          TagStructureMember "nToolLowerLimitValue"
          TagStructureMember "nToolUpperLimitValue"
          TagStructureMember "nDecimalPosition"
          TagStructureMember "nPitchPresentValueMAX/ColorAverageH (hue)"
          TagStructureMember "nPitchPresentValueMIN/ColorAverageS(saturation)"
          TagStructureMember "nNumberOfPitches/ColorAverageV(brightness)/BrightnessAverage"
          TagStructureMember "nReserved1"
        TagArrayMember "[30]"
          TagStructureMember "nToolMatchingRate"
          TagStructureMember "nToolMatchingRateMAX"
          TagStructureMember "nToolMatchingRateMIN"
          TagStructureMember "nToolLowerLimitValue"
          TagStructureMember "nToolUpperLimitValue"
          TagStructureMember "nDecimalPosition"
          TagStructureMember "nPitchPresentValueMAX/ColorAverageH (hue)"
          TagStructureMember "nPitchPresentValueMIN/ColorAverageS(saturation)"
          TagStructureMember "nNumberOfPitches/ColorAverageV(brightness)/BrightnessAverage"
          TagStructureMember "nReserved1"
        TagArrayMember "[31]"
          TagStructureMember "nToolMatchingRate"
          TagStructureMember "nToolMatchingRateMAX"
          TagStructureMember "nToolMatchingRateMIN"
          TagStructureMember "nToolLowerLimitValue"
          TagStructureMember "nToolUpperLimitValue"
          TagStructureMember "nDecimalPosition"
          TagStructureMember "nPitchPresentValueMAX/ColorAverageH (hue)"
          TagStructureMember "nPitchPresentValueMIN/ColorAverageS(saturation)"
          TagStructureMember "nNumberOfPitches/ColorAverageV(brightness)/BrightnessAverage"
          TagStructureMember "nReserved1"
        TagArrayMember "[32]"
          TagStructureMember "nToolMatchingRate"
          TagStructureMember "nToolMatchingRateMAX"
          TagStructureMember "nToolMatchingRateMIN"
          TagStructureMember "nToolLowerLimitValue"
          TagStructureMember "nToolUpperLimitValue"
          TagStructureMember "nDecimalPosition"
          TagStructureMember "nPitchPresentValueMAX/ColorAverageH (hue)"
          TagStructureMember "nPitchPresentValueMIN/ColorAverageS(saturation)"
          TagStructureMember "nNumberOfPitches/ColorAverageV(brightness)/BrightnessAverage"
          TagStructureMember "nReserved1"
        TagArrayMember "[33]"
          TagStructureMember "nToolMatchingRate"
          TagStructureMember "nToolMatchingRateMAX"
          TagStructureMember "nToolMatchingRateMIN"
          TagStructureMember "nToolLowerLimitValue"
          TagStructureMember "nToolUpperLimitValue"
          TagStructureMember "nDecimalPosition"
          TagStructureMember "nPitchPresentValueMAX/ColorAverageH (hue)"
          TagStructureMember "nPitchPresentValueMIN/ColorAverageS(saturation)"
          TagStructureMember "nNumberOfPitches/ColorAverageV(brightness)/BrightnessAverage"
          TagStructureMember "nReserved1"
        TagArrayMember "[34]"
          TagStructureMember "nToolMatchingRate"
          TagStructureMember "nToolMatchingRateMAX"
          TagStructureMember "nToolMatchingRateMIN"
          TagStructureMember "nToolLowerLimitValue"
          TagStructureMember "nToolUpperLimitValue"
          TagStructureMember "nDecimalPosition"
          TagStructureMember "nPitchPresentValueMAX/ColorAverageH (hue)"
          TagStructureMember "nPitchPresentValueMIN/ColorAverageS(saturation)"
          TagStructureMember "nNumberOfPitches/ColorAverageV(brightness)/BrightnessAverage"
          TagStructureMember "nReserved1"
        TagArrayMember "[35]"
          TagStructureMember "nToolMatchingRate"
          TagStructureMember "nToolMatchingRateMAX"
          TagStructureMember "nToolMatchingRateMIN"
          TagStructureMember "nToolLowerLimitValue"
          TagStructureMember "nToolUpperLimitValue"
          TagStructureMember "nDecimalPosition"
          TagStructureMember "nPitchPresentValueMAX/ColorAverageH (hue)"
          TagStructureMember "nPitchPresentValueMIN/ColorAverageS(saturation)"
          TagStructureMember "nNumberOfPitches/ColorAverageV(brightness)/BrightnessAverage"
          TagStructureMember "nReserved1"
        TagArrayMember "[36]"
          TagStructureMember "nToolMatchingRate"
          TagStructureMember "nToolMatchingRateMAX"
          TagStructureMember "nToolMatchingRateMIN"
          TagStructureMember "nToolLowerLimitValue"
          TagStructureMember "nToolUpperLimitValue"
          TagStructureMember "nDecimalPosition"
          TagStructureMember "nPitchPresentValueMAX/ColorAverageH (hue)"
          TagStructureMember "nPitchPresentValueMIN/ColorAverageS(saturation)"
          TagStructureMember "nNumberOfPitches/ColorAverageV(brightness)/BrightnessAverage"
          TagStructureMember "nReserved1"
        TagArrayMember "[37]"
          TagStructureMember "nToolMatchingRate"
          TagStructureMember "nToolMatchingRateMAX"
          TagStructureMember "nToolMatchingRateMIN"
          TagStructureMember "nToolLowerLimitValue"
          TagStructureMember "nToolUpperLimitValue"
          TagStructureMember "nDecimalPosition"
          TagStructureMember "nPitchPresentValueMAX/ColorAverageH (hue)"
          TagStructureMember "nPitchPresentValueMIN/ColorAverageS(saturation)"
          TagStructureMember "nNumberOfPitches/ColorAverageV(brightness)/BrightnessAverage"
          TagStructureMember "nReserved1"
        TagArrayMember "[38]"
          TagStructureMember "nToolMatchingRate"
          TagStructureMember "nToolMatchingRateMAX"
          TagStructureMember "nToolMatchingRateMIN"
          TagStructureMember "nToolLowerLimitValue"
          TagStructureMember "nToolUpperLimitValue"
          TagStructureMember "nDecimalPosition"
          TagStructureMember "nPitchPresentValueMAX/ColorAverageH (hue)"
          TagStructureMember "nPitchPresentValueMIN/ColorAverageS(saturation)"
          TagStructureMember "nNumberOfPitches/ColorAverageV(brightness)/BrightnessAverage"
          TagStructureMember "nReserved1"
        TagArrayMember "[39]"
          TagStructureMember "nToolMatchingRate"
          TagStructureMember "nToolMatchingRateMAX"
          TagStructureMember "nToolMatchingRateMIN"
          TagStructureMember "nToolLowerLimitValue"
          TagStructureMember "nToolUpperLimitValue"
          TagStructureMember "nDecimalPosition"
          TagStructureMember "nPitchPresentValueMAX/ColorAverageH (hue)"
          TagStructureMember "nPitchPresentValueMIN/ColorAverageS(saturation)"
          TagStructureMember "nNumberOfPitches/ColorAverageV(brightness)/BrightnessAverage"
          TagStructureMember "nReserved1"
        TagArrayMember "[40]"
          TagStructureMember "nToolMatchingRate"
          TagStructureMember "nToolMatchingRateMAX"
          TagStructureMember "nToolMatchingRateMIN"
          TagStructureMember "nToolLowerLimitValue"
          TagStructureMember "nToolUpperLimitValue"
          TagStructureMember "nDecimalPosition"
          TagStructureMember "nPitchPresentValueMAX/ColorAverageH (hue)"
          TagStructureMember "nPitchPresentValueMIN/ColorAverageS(saturation)"
          TagStructureMember "nNumberOfPitches/ColorAverageV(brightness)/BrightnessAverage"
          TagStructureMember "nReserved1"
        TagArrayMember "[41]"
          TagStructureMember "nToolMatchingRate"
          TagStructureMember "nToolMatchingRateMAX"
          TagStructureMember "nToolMatchingRateMIN"
          TagStructureMember "nToolLowerLimitValue"
          TagStructureMember "nToolUpperLimitValue"
          TagStructureMember "nDecimalPosition"
          TagStructureMember "nPitchPresentValueMAX/ColorAverageH (hue)"
          TagStructureMember "nPitchPresentValueMIN/ColorAverageS(saturation)"
          TagStructureMember "nNumberOfPitches/ColorAverageV(brightness)/BrightnessAverage"
          TagStructureMember "nReserved1"
        TagArrayMember "[42]"
          TagStructureMember "nToolMatchingRate"
          TagStructureMember "nToolMatchingRateMAX"
          TagStructureMember "nToolMatchingRateMIN"
          TagStructureMember "nToolLowerLimitValue"
          TagStructureMember "nToolUpperLimitValue"
          TagStructureMember "nDecimalPosition"
          TagStructureMember "nPitchPresentValueMAX/ColorAverageH (hue)"
          TagStructureMember "nPitchPresentValueMIN/ColorAverageS(saturation)"
          TagStructureMember "nNumberOfPitches/ColorAverageV(brightness)/BrightnessAverage"
          TagStructureMember "nReserved1"
        TagArrayMember "[43]"
          TagStructureMember "nToolMatchingRate"
          TagStructureMember "nToolMatchingRateMAX"
          TagStructureMember "nToolMatchingRateMIN"
          TagStructureMember "nToolLowerLimitValue"
          TagStructureMember "nToolUpperLimitValue"
          TagStructureMember "nDecimalPosition"
          TagStructureMember "nPitchPresentValueMAX/ColorAverageH (hue)"
          TagStructureMember "nPitchPresentValueMIN/ColorAverageS(saturation)"
          TagStructureMember "nNumberOfPitches/ColorAverageV(brightness)/BrightnessAverage"
          TagStructureMember "nReserved1"
        TagArrayMember "[44]"
          TagStructureMember "nToolMatchingRate"
          TagStructureMember "nToolMatchingRateMAX"
          TagStructureMember "nToolMatchingRateMIN"
          TagStructureMember "nToolLowerLimitValue"
          TagStructureMember "nToolUpperLimitValue"
          TagStructureMember "nDecimalPosition"
          TagStructureMember "nPitchPresentValueMAX/ColorAverageH (hue)"
          TagStructureMember "nPitchPresentValueMIN/ColorAverageS(saturation)"
          TagStructureMember "nNumberOfPitches/ColorAverageV(brightness)/BrightnessAverage"
          TagStructureMember "nReserved1"
        TagArrayMember "[45]"
          TagStructureMember "nToolMatchingRate"
          TagStructureMember "nToolMatchingRateMAX"
          TagStructureMember "nToolMatchingRateMIN"
          TagStructureMember "nToolLowerLimitValue"
          TagStructureMember "nToolUpperLimitValue"
          TagStructureMember "nDecimalPosition"
          TagStructureMember "nPitchPresentValueMAX/ColorAverageH (hue)"
          TagStructureMember "nPitchPresentValueMIN/ColorAverageS(saturation)"
          TagStructureMember "nNumberOfPitches/ColorAverageV(brightness)/BrightnessAverage"
          TagStructureMember "nReserved1"
        TagArrayMember "[46]"
          TagStructureMember "nToolMatchingRate"
          TagStructureMember "nToolMatchingRateMAX"
          TagStructureMember "nToolMatchingRateMIN"
          TagStructureMember "nToolLowerLimitValue"
          TagStructureMember "nToolUpperLimitValue"
          TagStructureMember "nDecimalPosition"
          TagStructureMember "nPitchPresentValueMAX/ColorAverageH (hue)"
          TagStructureMember "nPitchPresentValueMIN/ColorAverageS(saturation)"
          TagStructureMember "nNumberOfPitches/ColorAverageV(brightness)/BrightnessAverage"
          TagStructureMember "nReserved1"
        TagArrayMember "[47]"
          TagStructureMember "nToolMatchingRate"
          TagStructureMember "nToolMatchingRateMAX"
          TagStructureMember "nToolMatchingRateMIN"
          TagStructureMember "nToolLowerLimitValue"
          TagStructureMember "nToolUpperLimitValue"
          TagStructureMember "nDecimalPosition"
          TagStructureMember "nPitchPresentValueMAX/ColorAverageH (hue)"
          TagStructureMember "nPitchPresentValueMIN/ColorAverageS(saturation)"
          TagStructureMember "nNumberOfPitches/ColorAverageV(brightness)/BrightnessAverage"
          TagStructureMember "nReserved1"
        TagArrayMember "[48]"
          TagStructureMember "nToolMatchingRate"
          TagStructureMember "nToolMatchingRateMAX"
          TagStructureMember "nToolMatchingRateMIN"
          TagStructureMember "nToolLowerLimitValue"
          TagStructureMember "nToolUpperLimitValue"
          TagStructureMember "nDecimalPosition"
          TagStructureMember "nPitchPresentValueMAX/ColorAverageH (hue)"
          TagStructureMember "nPitchPresentValueMIN/ColorAverageS(saturation)"
          TagStructureMember "nNumberOfPitches/ColorAverageV(brightness)/BrightnessAverage"
          TagStructureMember "nReserved1"
        TagArrayMember "[49]"
          TagStructureMember "nToolMatchingRate"
          TagStructureMember "nToolMatchingRateMAX"
          TagStructureMember "nToolMatchingRateMIN"
          TagStructureMember "nToolLowerLimitValue"
          TagStructureMember "nToolUpperLimitValue"
          TagStructureMember "nDecimalPosition"
          TagStructureMember "nPitchPresentValueMAX/ColorAverageH (hue)"
          TagStructureMember "nPitchPresentValueMIN/ColorAverageS(saturation)"
          TagStructureMember "nNumberOfPitches/ColorAverageV(brightness)/BrightnessAverage"
          TagStructureMember "nReserved1"
        TagArrayMember "[50]"
          TagStructureMember "nToolMatchingRate"
          TagStructureMember "nToolMatchingRateMAX"
          TagStructureMember "nToolMatchingRateMIN"
          TagStructureMember "nToolLowerLimitValue"
          TagStructureMember "nToolUpperLimitValue"
          TagStructureMember "nDecimalPosition"
          TagStructureMember "nPitchPresentValueMAX/ColorAverageH (hue)"
          TagStructureMember "nPitchPresentValueMIN/ColorAverageS(saturation)"
          TagStructureMember "nNumberOfPitches/ColorAverageV(brightness)/BrightnessAverage"
          TagStructureMember "nReserved1"
        TagArrayMember "[51]"
          TagStructureMember "nToolMatchingRate"
          TagStructureMember "nToolMatchingRateMAX"
          TagStructureMember "nToolMatchingRateMIN"
          TagStructureMember "nToolLowerLimitValue"
          TagStructureMember "nToolUpperLimitValue"
          TagStructureMember "nDecimalPosition"
          TagStructureMember "nPitchPresentValueMAX/ColorAverageH (hue)"
          TagStructureMember "nPitchPresentValueMIN/ColorAverageS(saturation)"
          TagStructureMember "nNumberOfPitches/ColorAverageV(brightness)/BrightnessAverage"
          TagStructureMember "nReserved1"
        TagArrayMember "[52]"
          TagStructureMember "nToolMatchingRate"
          TagStructureMember "nToolMatchingRateMAX"
          TagStructureMember "nToolMatchingRateMIN"
          TagStructureMember "nToolLowerLimitValue"
          TagStructureMember "nToolUpperLimitValue"
          TagStructureMember "nDecimalPosition"
          TagStructureMember "nPitchPresentValueMAX/ColorAverageH (hue)"
          TagStructureMember "nPitchPresentValueMIN/ColorAverageS(saturation)"
          TagStructureMember "nNumberOfPitches/ColorAverageV(brightness)/BrightnessAverage"
          TagStructureMember "nReserved1"
        TagArrayMember "[53]"
          TagStructureMember "nToolMatchingRate"
          TagStructureMember "nToolMatchingRateMAX"
          TagStructureMember "nToolMatchingRateMIN"
          TagStructureMember "nToolLowerLimitValue"
          TagStructureMember "nToolUpperLimitValue"
          TagStructureMember "nDecimalPosition"
          TagStructureMember "nPitchPresentValueMAX/ColorAverageH (hue)"
          TagStructureMember "nPitchPresentValueMIN/ColorAverageS(saturation)"
          TagStructureMember "nNumberOfPitches/ColorAverageV(brightness)/BrightnessAverage"
          TagStructureMember "nReserved1"
        TagArrayMember "[54]"
          TagStructureMember "nToolMatchingRate"
          TagStructureMember "nToolMatchingRateMAX"
          TagStructureMember "nToolMatchingRateMIN"
          TagStructureMember "nToolLowerLimitValue"
          TagStructureMember "nToolUpperLimitValue"
          TagStructureMember "nDecimalPosition"
          TagStructureMember "nPitchPresentValueMAX/ColorAverageH (hue)"
          TagStructureMember "nPitchPresentValueMIN/ColorAverageS(saturation)"
          TagStructureMember "nNumberOfPitches/ColorAverageV(brightness)/BrightnessAverage"
          TagStructureMember "nReserved1"
        TagArrayMember "[55]"
          TagStructureMember "nToolMatchingRate"
          TagStructureMember "nToolMatchingRateMAX"
          TagStructureMember "nToolMatchingRateMIN"
          TagStructureMember "nToolLowerLimitValue"
          TagStructureMember "nToolUpperLimitValue"
          TagStructureMember "nDecimalPosition"
          TagStructureMember "nPitchPresentValueMAX/ColorAverageH (hue)"
          TagStructureMember "nPitchPresentValueMIN/ColorAverageS(saturation)"
          TagStructureMember "nNumberOfPitches/ColorAverageV(brightness)/BrightnessAverage"
          TagStructureMember "nReserved1"
        TagArrayMember "[56]"
          TagStructureMember "nToolMatchingRate"
          TagStructureMember "nToolMatchingRateMAX"
          TagStructureMember "nToolMatchingRateMIN"
          TagStructureMember "nToolLowerLimitValue"
          TagStructureMember "nToolUpperLimitValue"
          TagStructureMember "nDecimalPosition"
          TagStructureMember "nPitchPresentValueMAX/ColorAverageH (hue)"
          TagStructureMember "nPitchPresentValueMIN/ColorAverageS(saturation)"
          TagStructureMember "nNumberOfPitches/ColorAverageV(brightness)/BrightnessAverage"
          TagStructureMember "nReserved1"
        TagArrayMember "[57]"
          TagStructureMember "nToolMatchingRate"
          TagStructureMember "nToolMatchingRateMAX"
          TagStructureMember "nToolMatchingRateMIN"
          TagStructureMember "nToolLowerLimitValue"
          TagStructureMember "nToolUpperLimitValue"
          TagStructureMember "nDecimalPosition"
          TagStructureMember "nPitchPresentValueMAX/ColorAverageH (hue)"
          TagStructureMember "nPitchPresentValueMIN/ColorAverageS(saturation)"
          TagStructureMember "nNumberOfPitches/ColorAverageV(brightness)/BrightnessAverage"
          TagStructureMember "nReserved1"
        TagArrayMember "[58]"
          TagStructureMember "nToolMatchingRate"
          TagStructureMember "nToolMatchingRateMAX"
          TagStructureMember "nToolMatchingRateMIN"
          TagStructureMember "nToolLowerLimitValue"
          TagStructureMember "nToolUpperLimitValue"
          TagStructureMember "nDecimalPosition"
          TagStructureMember "nPitchPresentValueMAX/ColorAverageH (hue)"
          TagStructureMember "nPitchPresentValueMIN/ColorAverageS(saturation)"
          TagStructureMember "nNumberOfPitches/ColorAverageV(brightness)/BrightnessAverage"
          TagStructureMember "nReserved1"
        TagArrayMember "[59]"
          TagStructureMember "nToolMatchingRate"
          TagStructureMember "nToolMatchingRateMAX"
          TagStructureMember "nToolMatchingRateMIN"
          TagStructureMember "nToolLowerLimitValue"
          TagStructureMember "nToolUpperLimitValue"
          TagStructureMember "nDecimalPosition"
          TagStructureMember "nPitchPresentValueMAX/ColorAverageH (hue)"
          TagStructureMember "nPitchPresentValueMIN/ColorAverageS(saturation)"
          TagStructureMember "nNumberOfPitches/ColorAverageV(brightness)/BrightnessAverage"
          TagStructureMember "nReserved1"
        TagArrayMember "[60]"
          TagStructureMember "nToolMatchingRate"
          TagStructureMember "nToolMatchingRateMAX"
          TagStructureMember "nToolMatchingRateMIN"
          TagStructureMember "nToolLowerLimitValue"
          TagStructureMember "nToolUpperLimitValue"
          TagStructureMember "nDecimalPosition"
          TagStructureMember "nPitchPresentValueMAX/ColorAverageH (hue)"
          TagStructureMember "nPitchPresentValueMIN/ColorAverageS(saturation)"
          TagStructureMember "nNumberOfPitches/ColorAverageV(brightness)/BrightnessAverage"
          TagStructureMember "nReserved1"
        TagArrayMember "[61]"
          TagStructureMember "nToolMatchingRate"
          TagStructureMember "nToolMatchingRateMAX"
          TagStructureMember "nToolMatchingRateMIN"
          TagStructureMember "nToolLowerLimitValue"
          TagStructureMember "nToolUpperLimitValue"
          TagStructureMember "nDecimalPosition"
          TagStructureMember "nPitchPresentValueMAX/ColorAverageH (hue)"
          TagStructureMember "nPitchPresentValueMIN/ColorAverageS(saturation)"
          TagStructureMember "nNumberOfPitches/ColorAverageV(brightness)/BrightnessAverage"
          TagStructureMember "nReserved1"
        TagArrayMember "[62]"
          TagStructureMember "nToolMatchingRate"
          TagStructureMember "nToolMatchingRateMAX"
          TagStructureMember "nToolMatchingRateMIN"
          TagStructureMember "nToolLowerLimitValue"
          TagStructureMember "nToolUpperLimitValue"
          TagStructureMember "nDecimalPosition"
          TagStructureMember "nPitchPresentValueMAX/ColorAverageH (hue)"
          TagStructureMember "nPitchPresentValueMIN/ColorAverageS(saturation)"
          TagStructureMember "nNumberOfPitches/ColorAverageV(brightness)/BrightnessAverage"
          TagStructureMember "nReserved1"
        TagArrayMember "[63]"
          TagStructureMember "nToolMatchingRate"
          TagStructureMember "nToolMatchingRateMAX"
          TagStructureMember "nToolMatchingRateMIN"
          TagStructureMember "nToolLowerLimitValue"
          TagStructureMember "nToolUpperLimitValue"
          TagStructureMember "nDecimalPosition"
          TagStructureMember "nPitchPresentValueMAX/ColorAverageH (hue)"
          TagStructureMember "nPitchPresentValueMIN/ColorAverageS(saturation)"
          TagStructureMember "nNumberOfPitches/ColorAverageV(brightness)/BrightnessAverage"
          TagStructureMember "nReserved1"
      TagStructureMember "ExtendedDeviceResult"
        TagStructureMember "nMasterNumber"
        TagStructureMember "aToolResult"
          TagArrayMember "[0]"
          TagArrayMember "[1]"
          TagArrayMember "[2]"
          TagArrayMember "[3]"
          TagArrayMember "[4]"
          TagArrayMember "[5]"
          TagArrayMember "[6]"
          TagArrayMember "[7]"
          TagArrayMember "[8]"
          TagArrayMember "[9]"
          TagArrayMember "[10]"
          TagArrayMember "[11]"
          TagArrayMember "[12]"
          TagArrayMember "[13]"
          TagArrayMember "[14]"
          TagArrayMember "[15]"
          TagArrayMember "[16]"
          TagArrayMember "[17]"
          TagArrayMember "[18]"
          TagArrayMember "[19]"
          TagArrayMember "[20]"
          TagArrayMember "[21]"
          TagArrayMember "[22]"
          TagArrayMember "[23]"
          TagArrayMember "[24]"
          TagArrayMember "[25]"
          TagArrayMember "[26]"
          TagArrayMember "[27]"
          TagArrayMember "[28]"
          TagArrayMember "[29]"
          TagArrayMember "[30]"
          TagArrayMember "[31]"
          TagArrayMember "[32]"
          TagArrayMember "[33]"
          TagArrayMember "[34]"
          TagArrayMember "[35]"
          TagArrayMember "[36]"
          TagArrayMember "[37]"
          TagArrayMember "[38]"
          TagArrayMember "[39]"
          TagArrayMember "[40]"
          TagArrayMember "[41]"
          TagArrayMember "[42]"
          TagArrayMember "[43]"
          TagArrayMember "[44]"
          TagArrayMember "[45]"
          TagArrayMember "[46]"
          TagArrayMember "[47]"
    TagStructureMember "Out"
      TagStructureMember "CommandControl"
        TagStructureMember "bTriggerRequest"
        TagStructureMember "bMasterRegistrationRequest"
        TagStructureMember "bProgramSwitchingRequest"
        TagStructureMember "bWarningClearRequest"
        TagStructureMember "bStatisticsResetRequest"
        TagStructureMember "bBufferClearRequest"
        TagStructureMember "bSDCardSaveStopRequest"
        TagStructureMember "bParameterChangeRequest"
        TagStructureMember "nReserved1"
        TagStructureMember "bResultAcquisitionCompleteNotification"
        TagStructureMember "bReserved2"
        TagStructureMember "bReserved3"
        TagStructureMember "bReserved4"
        TagStructureMember "bReserved5"
        TagStructureMember "bReserved6"
        TagStructureMember "bReserved7"
        TagStructureMember "bReserved8"
        TagStructureMember "nReserved9"
        TagStructureMember "nProgramNo"
        TagStructureMember "nSetNumber"
        TagStructureMember "nSetParameter"
    TagStructureMember "Para"
      TagStructureMember "nInAdr1"
      TagStructureMember "nInAdr2"
      TagStructureMember "nInAdr3"
      TagStructureMember "nInAdr4"
      TagStructureMember "nInAdr5"
      TagStructureMember "nInAdr6"
      TagStructureMember "nInAdr7"
      TagStructureMember "nInAdr8"
      TagStructureMember "nInAdr9"
      TagStructureMember "nInAdr10"
      TagStructureMember "nInAdr11"
      TagStructureMember "nInAdr12"
      TagStructureMember "nInAdr13"
      TagStructureMember "nInAdr14"
      TagStructureMember "nInAdr15"
      TagStructureMember "nInAdr16"
      TagStructureMember "nInAdr17"
      TagStructureMember "nInAdr18"
      TagStructureMember "nInAdr19"
      TagStructureMember "nInAdr20"
      TagStructureMember "nInAdr21"
      TagStructureMember "nInAdr22"
      TagStructureMember "nInAdr23"
      TagStructureMember "nInAdr24"
      TagStructureMember "nInAdr25"
      TagStructureMember "nInAdr26"
      TagStructureMember "nInAdr27"
      TagStructureMember "nInAdr28"
      TagStructureMember "nInAdr29"
      TagStructureMember "nInAdr30"
      TagStructureMember "nInAdr31"
      TagStructureMember "nInAdr32"
      TagStructureMember "nInAdr33"
      TagStructureMember "nInAdr34"
      TagStructureMember "nInAdr35"
      TagStructureMember "nInAdr36"
      TagStructureMember "nInAdr37"
      TagStructureMember "nInAdr38"
      TagStructureMember "nInAdr39"
      TagStructureMember "nInAdr40"
      TagStructureMember "nInAdr41"
      TagStructureMember "nInAdr42"
      TagStructureMember "nInAdr43"
      TagStructureMember "nInAdr44"
      TagStructureMember "nInAdr45"
      TagStructureMember "nInAdr46"
      TagStructureMember "nInAdr47"
      TagStructureMember "nInAdr48"
      TagStructureMember "nInAdr49"
      TagStructureMember "nInAdr50"
      TagStructureMember "nInAdr51"
      TagStructureMember "nInAdr52"
      TagStructureMember "nInAdr53"
      TagStructureMember "nInAdr54"
      TagStructureMember "nInAdr55"
      TagStructureMember "nInAdr56"
      TagStructureMember "nInAdr57"
      TagStructureMember "nInAdr58"
      TagStructureMember "nInAdr59"
      TagStructureMember "nInAdr60"
      TagStructureMember "nInAdr61"
      TagStructureMember "nInAdr62"
      TagStructureMember "nInAdr63"
      TagStructureMember "nInAdr64"
      TagStructureMember "nInAdr65"
      TagStructureMember "nInAdr66"
      TagStructureMember "nInAdr67"
      TagStructureMember "nInAdr68"
      TagStructureMember "nInAdr69"
      TagStructureMember "nInAdr70"
      TagStructureMember "nOutAdr1"
      TagStructureMember "aToolResult"
        TagArrayMember "[0]"
        TagArrayMember "[1]"
        TagArrayMember "[2]"
        TagArrayMember "[3]"
        TagArrayMember "[4]"
        TagArrayMember "[5]"
        TagArrayMember "[6]"
        TagArrayMember "[7]"
        TagArrayMember "[8]"
        TagArrayMember "[9]"
        TagArrayMember "[10]"
        TagArrayMember "[11]"
        TagArrayMember "[12]"
        TagArrayMember "[13]"
        TagArrayMember "[14]"
        TagArrayMember "[15]"
        TagArrayMember "[16]"
        TagArrayMember "[17]"
        TagArrayMember "[18]"
        TagArrayMember "[19]"
        TagArrayMember "[20]"
        TagArrayMember "[21]"
        TagArrayMember "[22]"
        TagArrayMember "[23]"
        TagArrayMember "[24]"
        TagArrayMember "[25]"
        TagArrayMember "[26]"
        TagArrayMember "[27]"
        TagArrayMember "[28]"
        TagArrayMember "[29]"
        TagArrayMember "[30]"
        TagArrayMember "[31]"
        TagArrayMember "[32]"
        TagArrayMember "[33]"
        TagArrayMember "[34]"
        TagArrayMember "[35]"
        TagArrayMember "[36]"
        TagArrayMember "[37]"
        TagArrayMember "[38]"
        TagArrayMember "[39]"
        TagArrayMember "[40]"
        TagArrayMember "[41]"
        TagArrayMember "[42]"
        TagArrayMember "[43]"
        TagArrayMember "[44]"
        TagArrayMember "[45]"
        TagArrayMember "[46]"
        TagArrayMember "[47]"
        TagArrayMember "[48]"
        TagArrayMember "[49]"
        TagArrayMember "[50]"
        TagArrayMember "[51]"
        TagArrayMember "[52]"
        TagArrayMember "[53]"
        TagArrayMember "[54]"
        TagArrayMember "[55]"
        TagArrayMember "[56]"
        TagArrayMember "[57]"
        TagArrayMember "[58]"
        TagArrayMember "[59]"
        TagArrayMember "[60]"
        TagArrayMember "[61]"
        TagArrayMember "[62]"
        TagArrayMember "[63]"
      TagStructureMember "aToolResultHMI"
        TagArrayMember "[0]"
        TagArrayMember "[1]"
        TagArrayMember "[2]"
        TagArrayMember "[3]"
        TagArrayMember "[4]"
        TagArrayMember "[5]"
        TagArrayMember "[6]"
        TagArrayMember "[7]"
        TagArrayMember "[8]"
        TagArrayMember "[9]"
        TagArrayMember "[10]"
        TagArrayMember "[11]"
        TagArrayMember "[12]"
        TagArrayMember "[13]"
        TagArrayMember "[14]"
        TagArrayMember "[15]"
      TagStructureMember "ToolResult"
        TagArrayMember "[0]"
          TagStructureMember "nToolMatchingRate"
          TagStructureMember "nToolMatchingRateMAX"
          TagStructureMember "nToolMatchingRateMIN"
          TagStructureMember "nToolLowerLimitValue"
          TagStructureMember "nToolUpperLimitValue"
          TagStructureMember "nDecimalPosition"
          TagStructureMember "nPitchPresentValueMAX/ColorAverageH (hue)"
          TagStructureMember "nPitchPresentValueMIN/ColorAverageS(saturation)"
          TagStructureMember "nNumberOfPitches/ColorAverageV(brightness)/BrightnessAverage"
          TagStructureMember "nReserved1"
        TagArrayMember "[1]"
          TagStructureMember "nToolMatchingRate"
          TagStructureMember "nToolMatchingRateMAX"
          TagStructureMember "nToolMatchingRateMIN"
          TagStructureMember "nToolLowerLimitValue"
          TagStructureMember "nToolUpperLimitValue"
          TagStructureMember "nDecimalPosition"
          TagStructureMember "nPitchPresentValueMAX/ColorAverageH (hue)"
          TagStructureMember "nPitchPresentValueMIN/ColorAverageS(saturation)"
          TagStructureMember "nNumberOfPitches/ColorAverageV(brightness)/BrightnessAverage"
          TagStructureMember "nReserved1"
        TagArrayMember "[2]"
          TagStructureMember "nToolMatchingRate"
          TagStructureMember "nToolMatchingRateMAX"
          TagStructureMember "nToolMatchingRateMIN"
          TagStructureMember "nToolLowerLimitValue"
          TagStructureMember "nToolUpperLimitValue"
          TagStructureMember "nDecimalPosition"
          TagStructureMember "nPitchPresentValueMAX/ColorAverageH (hue)"
          TagStructureMember "nPitchPresentValueMIN/ColorAverageS(saturation)"
          TagStructureMember "nNumberOfPitches/ColorAverageV(brightness)/BrightnessAverage"
          TagStructureMember "nReserved1"
        TagArrayMember "[3]"
          TagStructureMember "nToolMatchingRate"
          TagStructureMember "nToolMatchingRateMAX"
          TagStructureMember "nToolMatchingRateMIN"
          TagStructureMember "nToolLowerLimitValue"
          TagStructureMember "nToolUpperLimitValue"
          TagStructureMember "nDecimalPosition"
          TagStructureMember "nPitchPresentValueMAX/ColorAverageH (hue)"
          TagStructureMember "nPitchPresentValueMIN/ColorAverageS(saturation)"
          TagStructureMember "nNumberOfPitches/ColorAverageV(brightness)/BrightnessAverage"
          TagStructureMember "nReserved1"
        TagArrayMember "[4]"
          TagStructureMember "nToolMatchingRate"
          TagStructureMember "nToolMatchingRateMAX"
          TagStructureMember "nToolMatchingRateMIN"
          TagStructureMember "nToolLowerLimitValue"
          TagStructureMember "nToolUpperLimitValue"
          TagStructureMember "nDecimalPosition"
          TagStructureMember "nPitchPresentValueMAX/ColorAverageH (hue)"
          TagStructureMember "nPitchPresentValueMIN/ColorAverageS(saturation)"
          TagStructureMember "nNumberOfPitches/ColorAverageV(brightness)/BrightnessAverage"
          TagStructureMember "nReserved1"
        TagArrayMember "[5]"
          TagStructureMember "nToolMatchingRate"
          TagStructureMember "nToolMatchingRateMAX"
          TagStructureMember "nToolMatchingRateMIN"
          TagStructureMember "nToolLowerLimitValue"
          TagStructureMember "nToolUpperLimitValue"
          TagStructureMember "nDecimalPosition"
          TagStructureMember "nPitchPresentValueMAX/ColorAverageH (hue)"
          TagStructureMember "nPitchPresentValueMIN/ColorAverageS(saturation)"
          TagStructureMember "nNumberOfPitches/ColorAverageV(brightness)/BrightnessAverage"
          TagStructureMember "nReserved1"
        TagArrayMember "[6]"
          TagStructureMember "nToolMatchingRate"
          TagStructureMember "nToolMatchingRateMAX"
          TagStructureMember "nToolMatchingRateMIN"
          TagStructureMember "nToolLowerLimitValue"
          TagStructureMember "nToolUpperLimitValue"
          TagStructureMember "nDecimalPosition"
          TagStructureMember "nPitchPresentValueMAX/ColorAverageH (hue)"
          TagStructureMember "nPitchPresentValueMIN/ColorAverageS(saturation)"
          TagStructureMember "nNumberOfPitches/ColorAverageV(brightness)/BrightnessAverage"
          TagStructureMember "nReserved1"
        TagArrayMember "[7]"
          TagStructureMember "nToolMatchingRate"
          TagStructureMember "nToolMatchingRateMAX"
          TagStructureMember "nToolMatchingRateMIN"
          TagStructureMember "nToolLowerLimitValue"
          TagStructureMember "nToolUpperLimitValue"
          TagStructureMember "nDecimalPosition"
          TagStructureMember "nPitchPresentValueMAX/ColorAverageH (hue)"
          TagStructureMember "nPitchPresentValueMIN/ColorAverageS(saturation)"
          TagStructureMember "nNumberOfPitches/ColorAverageV(brightness)/BrightnessAverage"
          TagStructureMember "nReserved1"
        TagArrayMember "[8]"
          TagStructureMember "nToolMatchingRate"
          TagStructureMember "nToolMatchingRateMAX"
          TagStructureMember "nToolMatchingRateMIN"
          TagStructureMember "nToolLowerLimitValue"
          TagStructureMember "nToolUpperLimitValue"
          TagStructureMember "nDecimalPosition"
          TagStructureMember "nPitchPresentValueMAX/ColorAverageH (hue)"
          TagStructureMember "nPitchPresentValueMIN/ColorAverageS(saturation)"
          TagStructureMember "nNumberOfPitches/ColorAverageV(brightness)/BrightnessAverage"
          TagStructureMember "nReserved1"
        TagArrayMember "[9]"
          TagStructureMember "nToolMatchingRate"
          TagStructureMember "nToolMatchingRateMAX"
          TagStructureMember "nToolMatchingRateMIN"
          TagStructureMember "nToolLowerLimitValue"
          TagStructureMember "nToolUpperLimitValue"
          TagStructureMember "nDecimalPosition"
          TagStructureMember "nPitchPresentValueMAX/ColorAverageH (hue)"
          TagStructureMember "nPitchPresentValueMIN/ColorAverageS(saturation)"
          TagStructureMember "nNumberOfPitches/ColorAverageV(brightness)/BrightnessAverage"
          TagStructureMember "nReserved1"
        TagArrayMember "[10]"
          TagStructureMember "nToolMatchingRate"
          TagStructureMember "nToolMatchingRateMAX"
          TagStructureMember "nToolMatchingRateMIN"
          TagStructureMember "nToolLowerLimitValue"
          TagStructureMember "nToolUpperLimitValue"
          TagStructureMember "nDecimalPosition"
          TagStructureMember "nPitchPresentValueMAX/ColorAverageH (hue)"
          TagStructureMember "nPitchPresentValueMIN/ColorAverageS(saturation)"
          TagStructureMember "nNumberOfPitches/ColorAverageV(brightness)/BrightnessAverage"
          TagStructureMember "nReserved1"
        TagArrayMember "[11]"
          TagStructureMember "nToolMatchingRate"
          TagStructureMember "nToolMatchingRateMAX"
          TagStructureMember "nToolMatchingRateMIN"
          TagStructureMember "nToolLowerLimitValue"
          TagStructureMember "nToolUpperLimitValue"
          TagStructureMember "nDecimalPosition"
          TagStructureMember "nPitchPresentValueMAX/ColorAverageH (hue)"
          TagStructureMember "nPitchPresentValueMIN/ColorAverageS(saturation)"
          TagStructureMember "nNumberOfPitches/ColorAverageV(brightness)/BrightnessAverage"
          TagStructureMember "nReserved1"
        TagArrayMember "[12]"
          TagStructureMember "nToolMatchingRate"
          TagStructureMember "nToolMatchingRateMAX"
          TagStructureMember "nToolMatchingRateMIN"
          TagStructureMember "nToolLowerLimitValue"
          TagStructureMember "nToolUpperLimitValue"
          TagStructureMember "nDecimalPosition"
          TagStructureMember "nPitchPresentValueMAX/ColorAverageH (hue)"
          TagStructureMember "nPitchPresentValueMIN/ColorAverageS(saturation)"
          TagStructureMember "nNumberOfPitches/ColorAverageV(brightness)/BrightnessAverage"
          TagStructureMember "nReserved1"
        TagArrayMember "[13]"
          TagStructureMember "nToolMatchingRate"
          TagStructureMember "nToolMatchingRateMAX"
          TagStructureMember "nToolMatchingRateMIN"
          TagStructureMember "nToolLowerLimitValue"
          TagStructureMember "nToolUpperLimitValue"
          TagStructureMember "nDecimalPosition"
          TagStructureMember "nPitchPresentValueMAX/ColorAverageH (hue)"
          TagStructureMember "nPitchPresentValueMIN/ColorAverageS(saturation)"
          TagStructureMember "nNumberOfPitches/ColorAverageV(brightness)/BrightnessAverage"
          TagStructureMember "nReserved1"
        TagArrayMember "[14]"
          TagStructureMember "nToolMatchingRate"
          TagStructureMember "nToolMatchingRateMAX"
          TagStructureMember "nToolMatchingRateMIN"
          TagStructureMember "nToolLowerLimitValue"
          TagStructureMember "nToolUpperLimitValue"
          TagStructureMember "nDecimalPosition"
          TagStructureMember "nPitchPresentValueMAX/ColorAverageH (hue)"
          TagStructureMember "nPitchPresentValueMIN/ColorAverageS(saturation)"
          TagStructureMember "nNumberOfPitches/ColorAverageV(brightness)/BrightnessAverage"
          TagStructureMember "nReserved1"
        TagArrayMember "[15]"
          TagStructureMember "nToolMatchingRate"
          TagStructureMember "nToolMatchingRateMAX"
          TagStructureMember "nToolMatchingRateMIN"
          TagStructureMember "nToolLowerLimitValue"
          TagStructureMember "nToolUpperLimitValue"
          TagStructureMember "nDecimalPosition"
          TagStructureMember "nPitchPresentValueMAX/ColorAverageH (hue)"
          TagStructureMember "nPitchPresentValueMIN/ColorAverageS(saturation)"
          TagStructureMember "nNumberOfPitches/ColorAverageV(brightness)/BrightnessAverage"
          TagStructureMember "nReserved1"
        TagArrayMember "[16]"
          TagStructureMember "nToolMatchingRate"
          TagStructureMember "nToolMatchingRateMAX"
          TagStructureMember "nToolMatchingRateMIN"
          TagStructureMember "nToolLowerLimitValue"
          TagStructureMember "nToolUpperLimitValue"
          TagStructureMember "nDecimalPosition"
          TagStructureMember "nPitchPresentValueMAX/ColorAverageH (hue)"
          TagStructureMember "nPitchPresentValueMIN/ColorAverageS(saturation)"
          TagStructureMember "nNumberOfPitches/ColorAverageV(brightness)/BrightnessAverage"
          TagStructureMember "nReserved1"
        TagArrayMember "[17]"
          TagStructureMember "nToolMatchingRate"
          TagStructureMember "nToolMatchingRateMAX"
          TagStructureMember "nToolMatchingRateMIN"
          TagStructureMember "nToolLowerLimitValue"
          TagStructureMember "nToolUpperLimitValue"
          TagStructureMember "nDecimalPosition"
          TagStructureMember "nPitchPresentValueMAX/ColorAverageH (hue)"
          TagStructureMember "nPitchPresentValueMIN/ColorAverageS(saturation)"
          TagStructureMember "nNumberOfPitches/ColorAverageV(brightness)/BrightnessAverage"
          TagStructureMember "nReserved1"
        TagArrayMember "[18]"
          TagStructureMember "nToolMatchingRate"
          TagStructureMember "nToolMatchingRateMAX"
          TagStructureMember "nToolMatchingRateMIN"
          TagStructureMember "nToolLowerLimitValue"
          TagStructureMember "nToolUpperLimitValue"
          TagStructureMember "nDecimalPosition"
          TagStructureMember "nPitchPresentValueMAX/ColorAverageH (hue)"
          TagStructureMember "nPitchPresentValueMIN/ColorAverageS(saturation)"
          TagStructureMember "nNumberOfPitches/ColorAverageV(brightness)/BrightnessAverage"
          TagStructureMember "nReserved1"
        TagArrayMember "[19]"
          TagStructureMember "nToolMatchingRate"
          TagStructureMember "nToolMatchingRateMAX"
          TagStructureMember "nToolMatchingRateMIN"
          TagStructureMember "nToolLowerLimitValue"
          TagStructureMember "nToolUpperLimitValue"
          TagStructureMember "nDecimalPosition"
          TagStructureMember "nPitchPresentValueMAX/ColorAverageH (hue)"
          TagStructureMember "nPitchPresentValueMIN/ColorAverageS(saturation)"
          TagStructureMember "nNumberOfPitches/ColorAverageV(brightness)/BrightnessAverage"
          TagStructureMember "nReserved1"
        TagArrayMember "[20]"
          TagStructureMember "nToolMatchingRate"
          TagStructureMember "nToolMatchingRateMAX"
          TagStructureMember "nToolMatchingRateMIN"
          TagStructureMember "nToolLowerLimitValue"
          TagStructureMember "nToolUpperLimitValue"
          TagStructureMember "nDecimalPosition"
          TagStructureMember "nPitchPresentValueMAX/ColorAverageH (hue)"
          TagStructureMember "nPitchPresentValueMIN/ColorAverageS(saturation)"
          TagStructureMember "nNumberOfPitches/ColorAverageV(brightness)/BrightnessAverage"
          TagStructureMember "nReserved1"
        TagArrayMember "[21]"
          TagStructureMember "nToolMatchingRate"
          TagStructureMember "nToolMatchingRateMAX"
          TagStructureMember "nToolMatchingRateMIN"
          TagStructureMember "nToolLowerLimitValue"
          TagStructureMember "nToolUpperLimitValue"
          TagStructureMember "nDecimalPosition"
          TagStructureMember "nPitchPresentValueMAX/ColorAverageH (hue)"
          TagStructureMember "nPitchPresentValueMIN/ColorAverageS(saturation)"
          TagStructureMember "nNumberOfPitches/ColorAverageV(brightness)/BrightnessAverage"
          TagStructureMember "nReserved1"
        TagArrayMember "[22]"
          TagStructureMember "nToolMatchingRate"
          TagStructureMember "nToolMatchingRateMAX"
          TagStructureMember "nToolMatchingRateMIN"
          TagStructureMember "nToolLowerLimitValue"
          TagStructureMember "nToolUpperLimitValue"
          TagStructureMember "nDecimalPosition"
          TagStructureMember "nPitchPresentValueMAX/ColorAverageH (hue)"
          TagStructureMember "nPitchPresentValueMIN/ColorAverageS(saturation)"
          TagStructureMember "nNumberOfPitches/ColorAverageV(brightness)/BrightnessAverage"
          TagStructureMember "nReserved1"
        TagArrayMember "[23]"
          TagStructureMember "nToolMatchingRate"
          TagStructureMember "nToolMatchingRateMAX"
          TagStructureMember "nToolMatchingRateMIN"
          TagStructureMember "nToolLowerLimitValue"
          TagStructureMember "nToolUpperLimitValue"
          TagStructureMember "nDecimalPosition"
          TagStructureMember "nPitchPresentValueMAX/ColorAverageH (hue)"
          TagStructureMember "nPitchPresentValueMIN/ColorAverageS(saturation)"
          TagStructureMember "nNumberOfPitches/ColorAverageV(brightness)/BrightnessAverage"
          TagStructureMember "nReserved1"
        TagArrayMember "[24]"
          TagStructureMember "nToolMatchingRate"
          TagStructureMember "nToolMatchingRateMAX"
          TagStructureMember "nToolMatchingRateMIN"
          TagStructureMember "nToolLowerLimitValue"
          TagStructureMember "nToolUpperLimitValue"
          TagStructureMember "nDecimalPosition"
          TagStructureMember "nPitchPresentValueMAX/ColorAverageH (hue)"
          TagStructureMember "nPitchPresentValueMIN/ColorAverageS(saturation)"
          TagStructureMember "nNumberOfPitches/ColorAverageV(brightness)/BrightnessAverage"
          TagStructureMember "nReserved1"
        TagArrayMember "[25]"
          TagStructureMember "nToolMatchingRate"
          TagStructureMember "nToolMatchingRateMAX"
          TagStructureMember "nToolMatchingRateMIN"
          TagStructureMember "nToolLowerLimitValue"
          TagStructureMember "nToolUpperLimitValue"
          TagStructureMember "nDecimalPosition"
          TagStructureMember "nPitchPresentValueMAX/ColorAverageH (hue)"
          TagStructureMember "nPitchPresentValueMIN/ColorAverageS(saturation)"
          TagStructureMember "nNumberOfPitches/ColorAverageV(brightness)/BrightnessAverage"
          TagStructureMember "nReserved1"
        TagArrayMember "[26]"
          TagStructureMember "nToolMatchingRate"
          TagStructureMember "nToolMatchingRateMAX"
          TagStructureMember "nToolMatchingRateMIN"
          TagStructureMember "nToolLowerLimitValue"
          TagStructureMember "nToolUpperLimitValue"
          TagStructureMember "nDecimalPosition"
          TagStructureMember "nPitchPresentValueMAX/ColorAverageH (hue)"
          TagStructureMember "nPitchPresentValueMIN/ColorAverageS(saturation)"
          TagStructureMember "nNumberOfPitches/ColorAverageV(brightness)/BrightnessAverage"
          TagStructureMember "nReserved1"
        TagArrayMember "[27]"
          TagStructureMember "nToolMatchingRate"
          TagStructureMember "nToolMatchingRateMAX"
          TagStructureMember "nToolMatchingRateMIN"
          TagStructureMember "nToolLowerLimitValue"
          TagStructureMember "nToolUpperLimitValue"
          TagStructureMember "nDecimalPosition"
          TagStructureMember "nPitchPresentValueMAX/ColorAverageH (hue)"
          TagStructureMember "nPitchPresentValueMIN/ColorAverageS(saturation)"
          TagStructureMember "nNumberOfPitches/ColorAverageV(brightness)/BrightnessAverage"
          TagStructureMember "nReserved1"
        TagArrayMember "[28]"
          TagStructureMember "nToolMatchingRate"
          TagStructureMember "nToolMatchingRateMAX"
          TagStructureMember "nToolMatchingRateMIN"
          TagStructureMember "nToolLowerLimitValue"
          TagStructureMember "nToolUpperLimitValue"
          TagStructureMember "nDecimalPosition"
          TagStructureMember "nPitchPresentValueMAX/ColorAverageH (hue)"
          TagStructureMember "nPitchPresentValueMIN/ColorAverageS(saturation)"
          TagStructureMember "nNumberOfPitches/ColorAverageV(brightness)/BrightnessAverage"
          TagStructureMember "nReserved1"
        TagArrayMember "[29]"
          TagStructureMember "nToolMatchingRate"
          TagStructureMember "nToolMatchingRateMAX"
          TagStructureMember "nToolMatchingRateMIN"
          TagStructureMember "nToolLowerLimitValue"
          TagStructureMember "nToolUpperLimitValue"
          TagStructureMember "nDecimalPosition"
          TagStructureMember "nPitchPresentValueMAX/ColorAverageH (hue)"
          TagStructureMember "nPitchPresentValueMIN/ColorAverageS(saturation)"
          TagStructureMember "nNumberOfPitches/ColorAverageV(brightness)/BrightnessAverage"
          TagStructureMember "nReserved1"
        TagArrayMember "[30]"
          TagStructureMember "nToolMatchingRate"
          TagStructureMember "nToolMatchingRateMAX"
          TagStructureMember "nToolMatchingRateMIN"
          TagStructureMember "nToolLowerLimitValue"
          TagStructureMember "nToolUpperLimitValue"
          TagStructureMember "nDecimalPosition"
          TagStructureMember "nPitchPresentValueMAX/ColorAverageH (hue)"
          TagStructureMember "nPitchPresentValueMIN/ColorAverageS(saturation)"
          TagStructureMember "nNumberOfPitches/ColorAverageV(brightness)/BrightnessAverage"
          TagStructureMember "nReserved1"
        TagArrayMember "[31]"
          TagStructureMember "nToolMatchingRate"
          TagStructureMember "nToolMatchingRateMAX"
          TagStructureMember "nToolMatchingRateMIN"
          TagStructureMember "nToolLowerLimitValue"
          TagStructureMember "nToolUpperLimitValue"
          TagStructureMember "nDecimalPosition"
          TagStructureMember "nPitchPresentValueMAX/ColorAverageH (hue)"
          TagStructureMember "nPitchPresentValueMIN/ColorAverageS(saturation)"
          TagStructureMember "nNumberOfPitches/ColorAverageV(brightness)/BrightnessAverage"
          TagStructureMember "nReserved1"
        TagArrayMember "[32]"
          TagStructureMember "nToolMatchingRate"
          TagStructureMember "nToolMatchingRateMAX"
          TagStructureMember "nToolMatchingRateMIN"
          TagStructureMember "nToolLowerLimitValue"
          TagStructureMember "nToolUpperLimitValue"
          TagStructureMember "nDecimalPosition"
          TagStructureMember "nPitchPresentValueMAX/ColorAverageH (hue)"
          TagStructureMember "nPitchPresentValueMIN/ColorAverageS(saturation)"
          TagStructureMember "nNumberOfPitches/ColorAverageV(brightness)/BrightnessAverage"
          TagStructureMember "nReserved1"
        TagArrayMember "[33]"
          TagStructureMember "nToolMatchingRate"
          TagStructureMember "nToolMatchingRateMAX"
          TagStructureMember "nToolMatchingRateMIN"
          TagStructureMember "nToolLowerLimitValue"
          TagStructureMember "nToolUpperLimitValue"
          TagStructureMember "nDecimalPosition"
          TagStructureMember "nPitchPresentValueMAX/ColorAverageH (hue)"
          TagStructureMember "nPitchPresentValueMIN/ColorAverageS(saturation)"
          TagStructureMember "nNumberOfPitches/ColorAverageV(brightness)/BrightnessAverage"
          TagStructureMember "nReserved1"
        TagArrayMember "[34]"
          TagStructureMember "nToolMatchingRate"
          TagStructureMember "nToolMatchingRateMAX"
          TagStructureMember "nToolMatchingRateMIN"
          TagStructureMember "nToolLowerLimitValue"
          TagStructureMember "nToolUpperLimitValue"
          TagStructureMember "nDecimalPosition"
          TagStructureMember "nPitchPresentValueMAX/ColorAverageH (hue)"
          TagStructureMember "nPitchPresentValueMIN/ColorAverageS(saturation)"
          TagStructureMember "nNumberOfPitches/ColorAverageV(brightness)/BrightnessAverage"
          TagStructureMember "nReserved1"
        TagArrayMember "[35]"
          TagStructureMember "nToolMatchingRate"
          TagStructureMember "nToolMatchingRateMAX"
          TagStructureMember "nToolMatchingRateMIN"
          TagStructureMember "nToolLowerLimitValue"
          TagStructureMember "nToolUpperLimitValue"
          TagStructureMember "nDecimalPosition"
          TagStructureMember "nPitchPresentValueMAX/ColorAverageH (hue)"
          TagStructureMember "nPitchPresentValueMIN/ColorAverageS(saturation)"
          TagStructureMember "nNumberOfPitches/ColorAverageV(brightness)/BrightnessAverage"
          TagStructureMember "nReserved1"
        TagArrayMember "[36]"
          TagStructureMember "nToolMatchingRate"
          TagStructureMember "nToolMatchingRateMAX"
          TagStructureMember "nToolMatchingRateMIN"
          TagStructureMember "nToolLowerLimitValue"
          TagStructureMember "nToolUpperLimitValue"
          TagStructureMember "nDecimalPosition"
          TagStructureMember "nPitchPresentValueMAX/ColorAverageH (hue)"
          TagStructureMember "nPitchPresentValueMIN/ColorAverageS(saturation)"
          TagStructureMember "nNumberOfPitches/ColorAverageV(brightness)/BrightnessAverage"
          TagStructureMember "nReserved1"
        TagArrayMember "[37]"
          TagStructureMember "nToolMatchingRate"
          TagStructureMember "nToolMatchingRateMAX"
          TagStructureMember "nToolMatchingRateMIN"
          TagStructureMember "nToolLowerLimitValue"
          TagStructureMember "nToolUpperLimitValue"
          TagStructureMember "nDecimalPosition"
          TagStructureMember "nPitchPresentValueMAX/ColorAverageH (hue)"
          TagStructureMember "nPitchPresentValueMIN/ColorAverageS(saturation)"
          TagStructureMember "nNumberOfPitches/ColorAverageV(brightness)/BrightnessAverage"
          TagStructureMember "nReserved1"
        TagArrayMember "[38]"
          TagStructureMember "nToolMatchingRate"
          TagStructureMember "nToolMatchingRateMAX"
          TagStructureMember "nToolMatchingRateMIN"
          TagStructureMember "nToolLowerLimitValue"
          TagStructureMember "nToolUpperLimitValue"
          TagStructureMember "nDecimalPosition"
          TagStructureMember "nPitchPresentValueMAX/ColorAverageH (hue)"
          TagStructureMember "nPitchPresentValueMIN/ColorAverageS(saturation)"
          TagStructureMember "nNumberOfPitches/ColorAverageV(brightness)/BrightnessAverage"
          TagStructureMember "nReserved1"
        TagArrayMember "[39]"
          TagStructureMember "nToolMatchingRate"
          TagStructureMember "nToolMatchingRateMAX"
          TagStructureMember "nToolMatchingRateMIN"
          TagStructureMember "nToolLowerLimitValue"
          TagStructureMember "nToolUpperLimitValue"
          TagStructureMember "nDecimalPosition"
          TagStructureMember "nPitchPresentValueMAX/ColorAverageH (hue)"
          TagStructureMember "nPitchPresentValueMIN/ColorAverageS(saturation)"
          TagStructureMember "nNumberOfPitches/ColorAverageV(brightness)/BrightnessAverage"
          TagStructureMember "nReserved1"
        TagArrayMember "[40]"
          TagStructureMember "nToolMatchingRate"
          TagStructureMember "nToolMatchingRateMAX"
          TagStructureMember "nToolMatchingRateMIN"
          TagStructureMember "nToolLowerLimitValue"
          TagStructureMember "nToolUpperLimitValue"
          TagStructureMember "nDecimalPosition"
          TagStructureMember "nPitchPresentValueMAX/ColorAverageH (hue)"
          TagStructureMember "nPitchPresentValueMIN/ColorAverageS(saturation)"
          TagStructureMember "nNumberOfPitches/ColorAverageV(brightness)/BrightnessAverage"
          TagStructureMember "nReserved1"
        TagArrayMember "[41]"
          TagStructureMember "nToolMatchingRate"
          TagStructureMember "nToolMatchingRateMAX"
          TagStructureMember "nToolMatchingRateMIN"
          TagStructureMember "nToolLowerLimitValue"
          TagStructureMember "nToolUpperLimitValue"
          TagStructureMember "nDecimalPosition"
          TagStructureMember "nPitchPresentValueMAX/ColorAverageH (hue)"
          TagStructureMember "nPitchPresentValueMIN/ColorAverageS(saturation)"
          TagStructureMember "nNumberOfPitches/ColorAverageV(brightness)/BrightnessAverage"
          TagStructureMember "nReserved1"
        TagArrayMember "[42]"
          TagStructureMember "nToolMatchingRate"
          TagStructureMember "nToolMatchingRateMAX"
          TagStructureMember "nToolMatchingRateMIN"
          TagStructureMember "nToolLowerLimitValue"
          TagStructureMember "nToolUpperLimitValue"
          TagStructureMember "nDecimalPosition"
          TagStructureMember "nPitchPresentValueMAX/ColorAverageH (hue)"
          TagStructureMember "nPitchPresentValueMIN/ColorAverageS(saturation)"
          TagStructureMember "nNumberOfPitches/ColorAverageV(brightness)/BrightnessAverage"
          TagStructureMember "nReserved1"
        TagArrayMember "[43]"
          TagStructureMember "nToolMatchingRate"
          TagStructureMember "nToolMatchingRateMAX"
          TagStructureMember "nToolMatchingRateMIN"
          TagStructureMember "nToolLowerLimitValue"
          TagStructureMember "nToolUpperLimitValue"
          TagStructureMember "nDecimalPosition"
          TagStructureMember "nPitchPresentValueMAX/ColorAverageH (hue)"
          TagStructureMember "nPitchPresentValueMIN/ColorAverageS(saturation)"
          TagStructureMember "nNumberOfPitches/ColorAverageV(brightness)/BrightnessAverage"
          TagStructureMember "nReserved1"
        TagArrayMember "[44]"
          TagStructureMember "nToolMatchingRate"
          TagStructureMember "nToolMatchingRateMAX"
          TagStructureMember "nToolMatchingRateMIN"
          TagStructureMember "nToolLowerLimitValue"
          TagStructureMember "nToolUpperLimitValue"
          TagStructureMember "nDecimalPosition"
          TagStructureMember "nPitchPresentValueMAX/ColorAverageH (hue)"
          TagStructureMember "nPitchPresentValueMIN/ColorAverageS(saturation)"
          TagStructureMember "nNumberOfPitches/ColorAverageV(brightness)/BrightnessAverage"
          TagStructureMember "nReserved1"
        TagArrayMember "[45]"
          TagStructureMember "nToolMatchingRate"
          TagStructureMember "nToolMatchingRateMAX"
          TagStructureMember "nToolMatchingRateMIN"
          TagStructureMember "nToolLowerLimitValue"
          TagStructureMember "nToolUpperLimitValue"
          TagStructureMember "nDecimalPosition"
          TagStructureMember "nPitchPresentValueMAX/ColorAverageH (hue)"
          TagStructureMember "nPitchPresentValueMIN/ColorAverageS(saturation)"
          TagStructureMember "nNumberOfPitches/ColorAverageV(brightness)/BrightnessAverage"
          TagStructureMember "nReserved1"
        TagArrayMember "[46]"
          TagStructureMember "nToolMatchingRate"
          TagStructureMember "nToolMatchingRateMAX"
          TagStructureMember "nToolMatchingRateMIN"
          TagStructureMember "nToolLowerLimitValue"
          TagStructureMember "nToolUpperLimitValue"
          TagStructureMember "nDecimalPosition"
          TagStructureMember "nPitchPresentValueMAX/ColorAverageH (hue)"
          TagStructureMember "nPitchPresentValueMIN/ColorAverageS(saturation)"
          TagStructureMember "nNumberOfPitches/ColorAverageV(brightness)/BrightnessAverage"
          TagStructureMember "nReserved1"
        TagArrayMember "[47]"
          TagStructureMember "nToolMatchingRate"
          TagStructureMember "nToolMatchingRateMAX"
          TagStructureMember "nToolMatchingRateMIN"
          TagStructureMember "nToolLowerLimitValue"
          TagStructureMember "nToolUpperLimitValue"
          TagStructureMember "nDecimalPosition"
          TagStructureMember "nPitchPresentValueMAX/ColorAverageH (hue)"
          TagStructureMember "nPitchPresentValueMIN/ColorAverageS(saturation)"
          TagStructureMember "nNumberOfPitches/ColorAverageV(brightness)/BrightnessAverage"
          TagStructureMember "nReserved1"
        TagArrayMember "[48]"
          TagStructureMember "nToolMatchingRate"
          TagStructureMember "nToolMatchingRateMAX"
          TagStructureMember "nToolMatchingRateMIN"
          TagStructureMember "nToolLowerLimitValue"
          TagStructureMember "nToolUpperLimitValue"
          TagStructureMember "nDecimalPosition"
          TagStructureMember "nPitchPresentValueMAX/ColorAverageH (hue)"
          TagStructureMember "nPitchPresentValueMIN/ColorAverageS(saturation)"
          TagStructureMember "nNumberOfPitches/ColorAverageV(brightness)/BrightnessAverage"
          TagStructureMember "nReserved1"
        TagArrayMember "[49]"
          TagStructureMember "nToolMatchingRate"
          TagStructureMember "nToolMatchingRateMAX"
          TagStructureMember "nToolMatchingRateMIN"
          TagStructureMember "nToolLowerLimitValue"
          TagStructureMember "nToolUpperLimitValue"
          TagStructureMember "nDecimalPosition"
          TagStructureMember "nPitchPresentValueMAX/ColorAverageH (hue)"
          TagStructureMember "nPitchPresentValueMIN/ColorAverageS(saturation)"
          TagStructureMember "nNumberOfPitches/ColorAverageV(brightness)/BrightnessAverage"
          TagStructureMember "nReserved1"
        TagArrayMember "[50]"
          TagStructureMember "nToolMatchingRate"
          TagStructureMember "nToolMatchingRateMAX"
          TagStructureMember "nToolMatchingRateMIN"
          TagStructureMember "nToolLowerLimitValue"
          TagStructureMember "nToolUpperLimitValue"
          TagStructureMember "nDecimalPosition"
          TagStructureMember "nPitchPresentValueMAX/ColorAverageH (hue)"
          TagStructureMember "nPitchPresentValueMIN/ColorAverageS(saturation)"
          TagStructureMember "nNumberOfPitches/ColorAverageV(brightness)/BrightnessAverage"
          TagStructureMember "nReserved1"
        TagArrayMember "[51]"
          TagStructureMember "nToolMatchingRate"
          TagStructureMember "nToolMatchingRateMAX"
          TagStructureMember "nToolMatchingRateMIN"
          TagStructureMember "nToolLowerLimitValue"
          TagStructureMember "nToolUpperLimitValue"
          TagStructureMember "nDecimalPosition"
          TagStructureMember "nPitchPresentValueMAX/ColorAverageH (hue)"
          TagStructureMember "nPitchPresentValueMIN/ColorAverageS(saturation)"
          TagStructureMember "nNumberOfPitches/ColorAverageV(brightness)/BrightnessAverage"
          TagStructureMember "nReserved1"
        TagArrayMember "[52]"
          TagStructureMember "nToolMatchingRate"
          TagStructureMember "nToolMatchingRateMAX"
          TagStructureMember "nToolMatchingRateMIN"
          TagStructureMember "nToolLowerLimitValue"
          TagStructureMember "nToolUpperLimitValue"
          TagStructureMember "nDecimalPosition"
          TagStructureMember "nPitchPresentValueMAX/ColorAverageH (hue)"
          TagStructureMember "nPitchPresentValueMIN/ColorAverageS(saturation)"
          TagStructureMember "nNumberOfPitches/ColorAverageV(brightness)/BrightnessAverage"
          TagStructureMember "nReserved1"
        TagArrayMember "[53]"
          TagStructureMember "nToolMatchingRate"
          TagStructureMember "nToolMatchingRateMAX"
          TagStructureMember "nToolMatchingRateMIN"
          TagStructureMember "nToolLowerLimitValue"
          TagStructureMember "nToolUpperLimitValue"
          TagStructureMember "nDecimalPosition"
          TagStructureMember "nPitchPresentValueMAX/ColorAverageH (hue)"
          TagStructureMember "nPitchPresentValueMIN/ColorAverageS(saturation)"
          TagStructureMember "nNumberOfPitches/ColorAverageV(brightness)/BrightnessAverage"
          TagStructureMember "nReserved1"
        TagArrayMember "[54]"
          TagStructureMember "nToolMatchingRate"
          TagStructureMember "nToolMatchingRateMAX"
          TagStructureMember "nToolMatchingRateMIN"
          TagStructureMember "nToolLowerLimitValue"
          TagStructureMember "nToolUpperLimitValue"
          TagStructureMember "nDecimalPosition"
          TagStructureMember "nPitchPresentValueMAX/ColorAverageH (hue)"
          TagStructureMember "nPitchPresentValueMIN/ColorAverageS(saturation)"
          TagStructureMember "nNumberOfPitches/ColorAverageV(brightness)/BrightnessAverage"
          TagStructureMember "nReserved1"
        TagArrayMember "[55]"
          TagStructureMember "nToolMatchingRate"
          TagStructureMember "nToolMatchingRateMAX"
          TagStructureMember "nToolMatchingRateMIN"
          TagStructureMember "nToolLowerLimitValue"
          TagStructureMember "nToolUpperLimitValue"
          TagStructureMember "nDecimalPosition"
          TagStructureMember "nPitchPresentValueMAX/ColorAverageH (hue)"
          TagStructureMember "nPitchPresentValueMIN/ColorAverageS(saturation)"
          TagStructureMember "nNumberOfPitches/ColorAverageV(brightness)/BrightnessAverage"
          TagStructureMember "nReserved1"
        TagArrayMember "[56]"
          TagStructureMember "nToolMatchingRate"
          TagStructureMember "nToolMatchingRateMAX"
          TagStructureMember "nToolMatchingRateMIN"
          TagStructureMember "nToolLowerLimitValue"
          TagStructureMember "nToolUpperLimitValue"
          TagStructureMember "nDecimalPosition"
          TagStructureMember "nPitchPresentValueMAX/ColorAverageH (hue)"
          TagStructureMember "nPitchPresentValueMIN/ColorAverageS(saturation)"
          TagStructureMember "nNumberOfPitches/ColorAverageV(brightness)/BrightnessAverage"
          TagStructureMember "nReserved1"
        TagArrayMember "[57]"
          TagStructureMember "nToolMatchingRate"
          TagStructureMember "nToolMatchingRateMAX"
          TagStructureMember "nToolMatchingRateMIN"
          TagStructureMember "nToolLowerLimitValue"
          TagStructureMember "nToolUpperLimitValue"
          TagStructureMember "nDecimalPosition"
          TagStructureMember "nPitchPresentValueMAX/ColorAverageH (hue)"
          TagStructureMember "nPitchPresentValueMIN/ColorAverageS(saturation)"
          TagStructureMember "nNumberOfPitches/ColorAverageV(brightness)/BrightnessAverage"
          TagStructureMember "nReserved1"
        TagArrayMember "[58]"
          TagStructureMember "nToolMatchingRate"
          TagStructureMember "nToolMatchingRateMAX"
          TagStructureMember "nToolMatchingRateMIN"
          TagStructureMember "nToolLowerLimitValue"
          TagStructureMember "nToolUpperLimitValue"
          TagStructureMember "nDecimalPosition"
          TagStructureMember "nPitchPresentValueMAX/ColorAverageH (hue)"
          TagStructureMember "nPitchPresentValueMIN/ColorAverageS(saturation)"
          TagStructureMember "nNumberOfPitches/ColorAverageV(brightness)/BrightnessAverage"
          TagStructureMember "nReserved1"
        TagArrayMember "[59]"
          TagStructureMember "nToolMatchingRate"
          TagStructureMember "nToolMatchingRateMAX"
          TagStructureMember "nToolMatchingRateMIN"
          TagStructureMember "nToolLowerLimitValue"
          TagStructureMember "nToolUpperLimitValue"
          TagStructureMember "nDecimalPosition"
          TagStructureMember "nPitchPresentValueMAX/ColorAverageH (hue)"
          TagStructureMember "nPitchPresentValueMIN/ColorAverageS(saturation)"
          TagStructureMember "nNumberOfPitches/ColorAverageV(brightness)/BrightnessAverage"
          TagStructureMember "nReserved1"
        TagArrayMember "[60]"
          TagStructureMember "nToolMatchingRate"
          TagStructureMember "nToolMatchingRateMAX"
          TagStructureMember "nToolMatchingRateMIN"
          TagStructureMember "nToolLowerLimitValue"
          TagStructureMember "nToolUpperLimitValue"
          TagStructureMember "nDecimalPosition"
          TagStructureMember "nPitchPresentValueMAX/ColorAverageH (hue)"
          TagStructureMember "nPitchPresentValueMIN/ColorAverageS(saturation)"
          TagStructureMember "nNumberOfPitches/ColorAverageV(brightness)/BrightnessAverage"
          TagStructureMember "nReserved1"
        TagArrayMember "[61]"
          TagStructureMember "nToolMatchingRate"
          TagStructureMember "nToolMatchingRateMAX"
          TagStructureMember "nToolMatchingRateMIN"
          TagStructureMember "nToolLowerLimitValue"
          TagStructureMember "nToolUpperLimitValue"
          TagStructureMember "nDecimalPosition"
          TagStructureMember "nPitchPresentValueMAX/ColorAverageH (hue)"
          TagStructureMember "nPitchPresentValueMIN/ColorAverageS(saturation)"
          TagStructureMember "nNumberOfPitches/ColorAverageV(brightness)/BrightnessAverage"
          TagStructureMember "nReserved1"
        TagArrayMember "[62]"
          TagStructureMember "nToolMatchingRate"
          TagStructureMember "nToolMatchingRateMAX"
          TagStructureMember "nToolMatchingRateMIN"
          TagStructureMember "nToolLowerLimitValue"
          TagStructureMember "nToolUpperLimitValue"
          TagStructureMember "nDecimalPosition"
          TagStructureMember "nPitchPresentValueMAX/ColorAverageH (hue)"
          TagStructureMember "nPitchPresentValueMIN/ColorAverageS(saturation)"
          TagStructureMember "nNumberOfPitches/ColorAverageV(brightness)/BrightnessAverage"
          TagStructureMember "nReserved1"
        TagArrayMember "[63]"
          TagStructureMember "nToolMatchingRate"
          TagStructureMember "nToolMatchingRateMAX"
          TagStructureMember "nToolMatchingRateMIN"
          TagStructureMember "nToolLowerLimitValue"
          TagStructureMember "nToolUpperLimitValue"
          TagStructureMember "nDecimalPosition"
          TagStructureMember "nPitchPresentValueMAX/ColorAverageH (hue)"
          TagStructureMember "nPitchPresentValueMIN/ColorAverageS(saturation)"
          TagStructureMember "nNumberOfPitches/ColorAverageV(brightness)/BrightnessAverage"
          TagStructureMember "nReserved1"
      TagStructureMember "nProgramNo"
      TagStructureMember "bProductOverallOK"
      TagStructureMember "bProductOverallNG"
